Staubli VAL3: remErrBusy.pgx

program remErrBusy(string& sReturn[] (dimensions=1))
begin
  // Error raised when Remote Motion task is busy
  //
  logMsg("call remErrBusy")
  sReturn="ERROR 201"
  sReturn=sReturn+": Move command already active."
  putln(sReturn)
  logMsg(sReturn)
end
